// SIMATIC S7-200 project (STEP 7-Micro/WIN), CPU 224 REL 02.01

ORGANIZATION_BLOCK MAIN:OB1
TITLE=PROGRAM COMMENTS
BEGIN
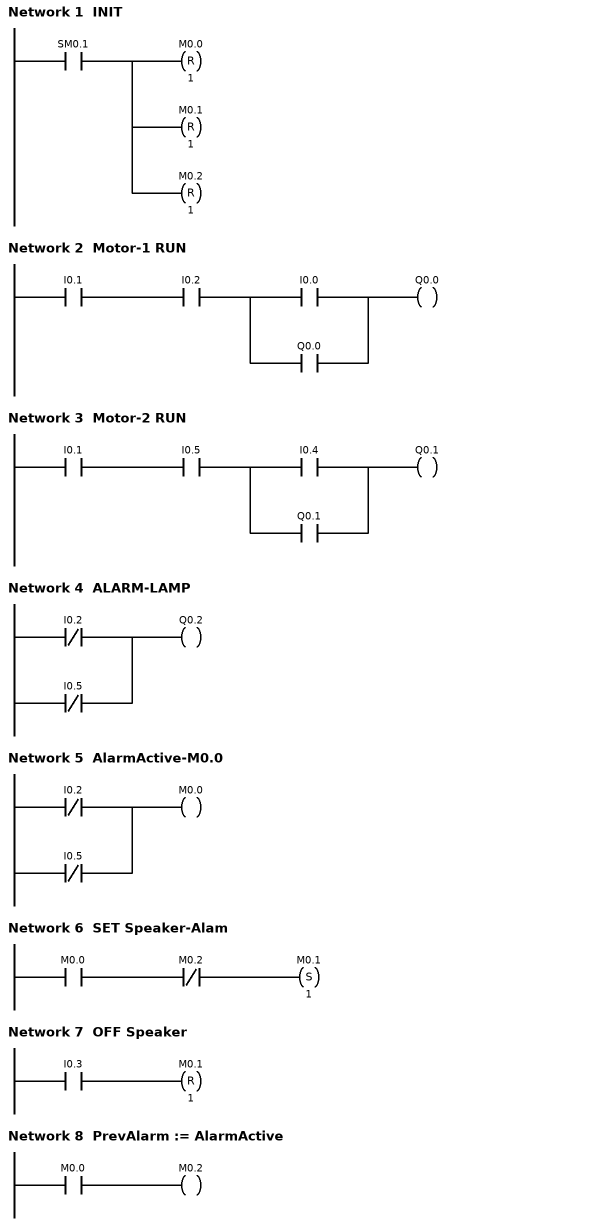
Network 1 // INIT
LD     SM0.1
R      M0.0, 1
R      M0.1, 1
R      M0.2, 1
Network 2 // Motor-1 RUN
LD     I0.1
A      I0.2
LD     I0.0
O      Q0.0
ALD
=      Q0.0
Network 3 // Motor-2 RUN
LD     I0.1
A      I0.5
LD     I0.4
O      Q0.1
ALD
=      Q0.1
Network 4 // ALARM-LAMP
LDN    I0.2
ON     I0.5
=      Q0.2
Network 5 // AlarmActive-M0.0
LDN    I0.2
ON     I0.5
=      M0.0
Network 6 // SET Speaker-Alam
LD     M0.0
AN     M0.2
S      M0.1, 1
Network 7 // OFF Speaker
LD     I0.3
R      M0.1, 1
Network 8 // PrevAlarm := AlarmActive
LD     M0.0
=      M0.2
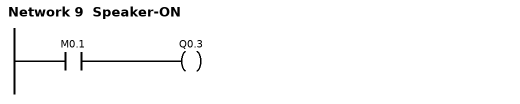
Network 9 // Speaker-ON
LD     M0.1
=      Q0.3
END_ORGANIZATION_BLOCK
